(* Schneider Machine Expert - Basic project resolucao, file version 2.7.0.0 *)
(* ProjectInformations: Name=Novo projeto *)

HARDWARE
  Cpu 0: TM221CE24R
  EthernetConfiguration: NetworkName=M221, IpAllocationMode=FixedAddress, IpAddress=0.0.0.0, SubnetMask=0.0.0.0
  SerialLineConfiguration: Baud=Baud19200, Parity=ParityEven, DataBits=DataBits8, StopBits=StopBits1, PhysicalMedium=PhysicalMediumRs485, TransmissionMode=TransmissionModeModbusRtu, SlaveId=1, Addressing=SlaveAddressing
  MastTask: UsePeriodScanMode=false, PeriodScan=100
  FastTask: Period=255
  CpuBehavior: StartingMode=StartAsPreviousState, AutoSaveRamOnEeprom=true, WatchdogPeriod=250

SYMBOLS  (address, symbol, comment, settings)
  %M0       SIG_IN_BOT_1
  %M1       SIG_BOR
  %M2       SIG_OUT_PUL_1
  %I0.0     IN_BOT_1
  %Q0.1     OUT_PUL_1

POU Entradas
  (* SectionNumber=1 *)

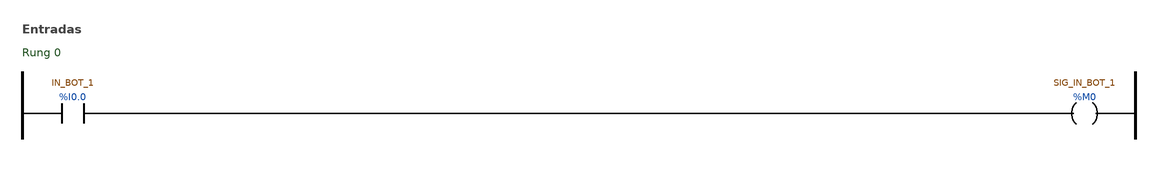

// Rung 0
  LD %I0.0                (* IN_BOT_1 *)
  ST %M0                  (* SIG_IN_BOT_1 *)
  // as ST:
  //   SIG_IN_BOT_1 := IN_BOT_1;

POU Lógicas
  (* SectionNumber=2 *)

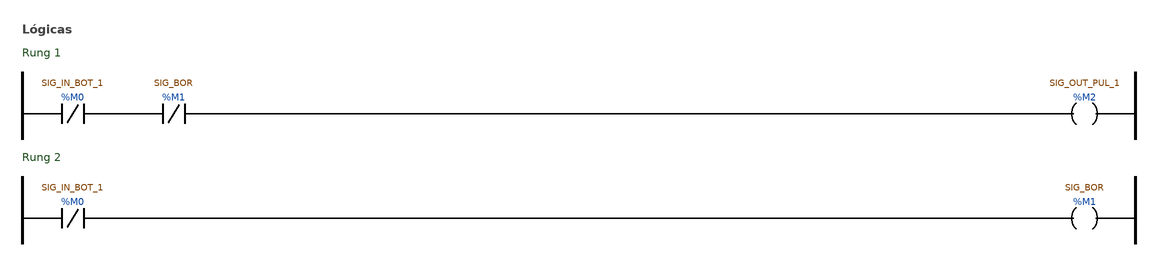

// Rung 1
  LDN %M0                 (* SIG_IN_BOT_1 *)
  ANDN %M1                (* SIG_BOR *)
  ST %M2                  (* SIG_OUT_PUL_1 *)
  // as ST:
  //   SIG_OUT_PUL_1 := NOT SIG_IN_BOT_1 AND NOT SIG_BOR;

// Rung 2
  LDN %M0                 (* SIG_IN_BOT_1 *)
  ST %M1                  (* SIG_BOR *)
  // as ST:
  //   SIG_BOR := NOT SIG_IN_BOT_1;

POU Saídas
  (* SectionNumber=3 *)

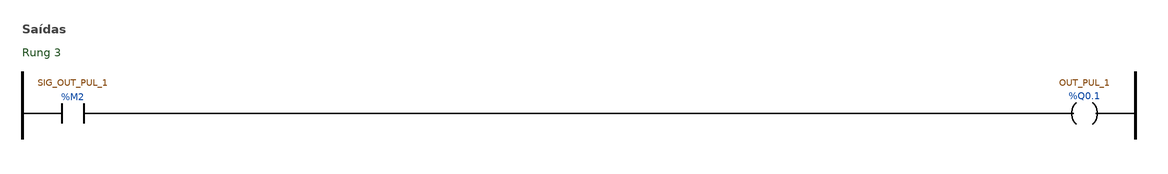

// Rung 3
  LD %M2                  (* SIG_OUT_PUL_1 *)
  ST %Q0.1                (* OUT_PUL_1 *)
  // as ST:
  //   OUT_PUL_1 := SIG_OUT_PUL_1;
